// Mitsubishi GX Works2 project: solvvNpress_3   PLC: Q03UDV

PROGRAM MAIN
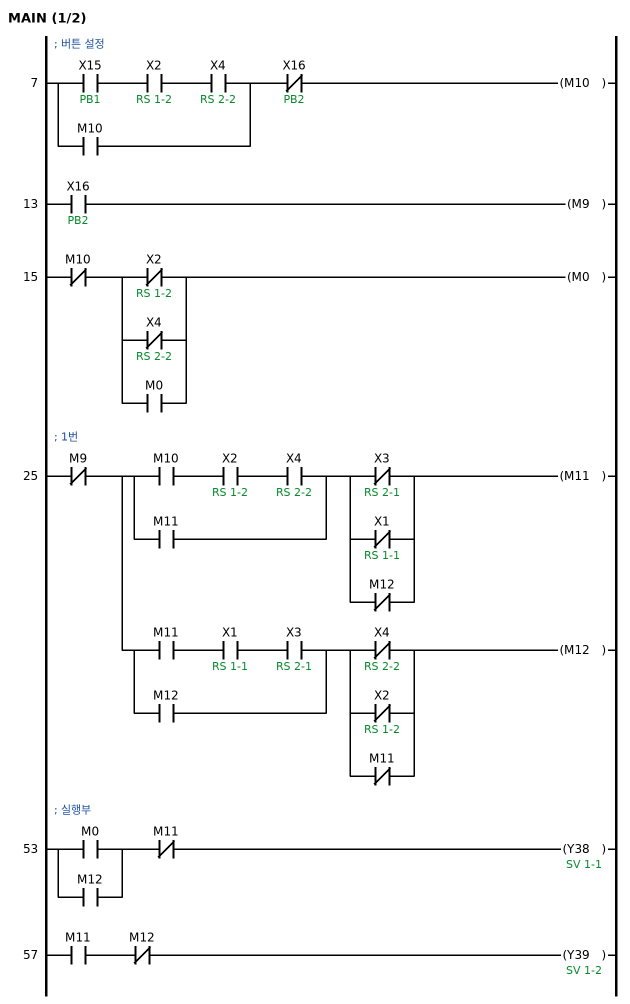
; 버튼 설정
7     LD      X15  ; PB1
      AND     X2  ; RS 1-2
      AND     X4  ; RS 2-2
      OR      M10
      ANI     X16  ; PB2
      OUT     M10
13    LD      X16  ; PB2
      OUT     M9
15    LDI     M10
      LDI     X2  ; RS 1-2
      ORI     X4  ; RS 2-2
      OR      M0
      ANB
      OUT     M0
; 1번
25    LDI     M9
      MPS
      LD      M10
      AND     X2  ; RS 1-2
      AND     X4  ; RS 2-2
      OR      M11
      ANB
      LDI     X3  ; RS 2-1
      ORI     X1  ; RS 1-1
      ORI     M12
      ANB
      OUT     M11
      MPP
      LD      M11
      AND     X1  ; RS 1-1
      AND     X3  ; RS 2-1
      OR      M12
      ANB
      LDI     X4  ; RS 2-2
      ORI     X2  ; RS 1-2
      ORI     M11
      ANB
      OUT     M12
; 실행부
53    LD      M0
      OR      M12
      ANI     M11
      OUT     Y38  ; SV 1-1
57    LD      M11
      ANI     M12
      OUT     Y39  ; SV 1-2
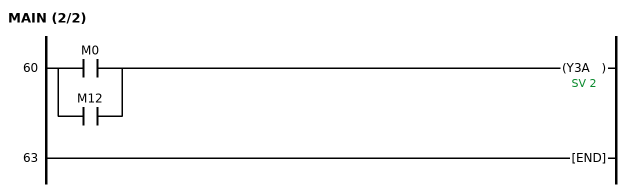
60    LD      M0
      OR      M12
      OUT     Y3A  ; SV 2
63    END
END_PROGRAM

// device comments not shown above
X17  ; PB3
X18  ; PB4
X19  ; PB5
Y30  ; LAMP1
Y31  ; LAMP2
Y3B  ; SV 3
